FUNCTION UpdateTimeStamp 
VAR_INPUT
	stUser : REFERENCE TO ST_USER;
END_VAR
VAR
	fbGETSYSTEMTIME : GETSYSTEMTIME;
	
	stFileTime : T_FILETIME;
END_VAR


fbGETSYSTEMTIME(timeLoDW =>stFileTime.dwLowDateTime ,
				timeHiDW =>stFileTime.dwHighDateTime );
				
stUser.dtTIME_STAMP:= FILETIME_TO_DT(fileTime := stFileTime);

END_FUNCTION

(* stored: Version 1.1.0.1, ProductVersion 3.1.4024.11
   POU UpdateTimeStamp: Id {3ebf2d11-b075-4b1e-bfc5-6a6be67fc618}, SpecialFunc None *)
